FUNCTION_BLOCK Sensor_MDL
  (* Version 1.0, 2005-11-13, Goran Cengic, Chalmers *)
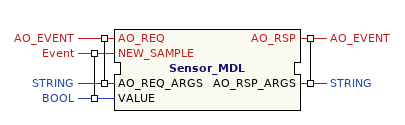
  EVENT_INPUT
    AO_REQ : AO_EVENT WITH AO_REQ_ARGS;
    NEW_SAMPLE WITH VALUE;
  END_EVENT
  EVENT_OUTPUT
    AO_RSP : AO_EVENT WITH AO_RSP_ARGS;
  END_EVENT
  VAR_INPUT
    AO_REQ_ARGS : STRING;
    VALUE : BOOL;
  END_VAR
  VAR_OUTPUT
    AO_RSP_ARGS : STRING;
  END_VAR
  VAR
    curValue : BOOL;
  END_VAR
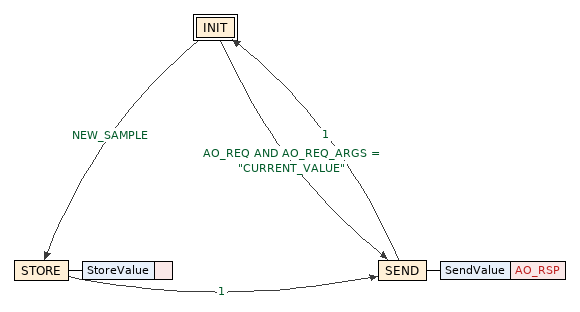
  EC_STATES
    INIT;
    SEND : SendValue -> AO_RSP;
    STORE : StoreValue;
  END_STATES
  EC_TRANSITIONS
    INIT TO SEND := AO_REQ AND AO_REQ_ARGS = "CURRENT_VALUE";
    SEND TO INIT := 1;
    INIT TO STORE := NEW_SAMPLE;
    STORE TO SEND := 1;
  END_TRANSITIONS
  ALGORITHM SendValue IN Java:
	    AO_RSP_ARGS = "CURRENT_VALUE " + curValue.toString();
  END_ALGORITHM
  ALGORITHM StoreValue IN Java:
	    curValue = VALUE;
  END_ALGORITHM
END_FUNCTION_BLOCK
